PROGRAM ReactorLevelAndPressureController
VAR_INPUT
	serialCommData : ST_SerialCommReadData;
	stop : BOOL;
	levelHigh : BOOL;
END_VAR
VAR_OUTPUT
	slurryInletValve : BOOL;
	slurryOutletValve : BOOL;
	extractiveOutletOnOffValve : BOOL;
	extractiveOutletControlValveClose : BOOL;
	extractiveOutletControlValveOpen : BOOL;
END_VAR
VAR
	
	// Handlers to call
	HandlePressureSensorScaling : PressureSensorScalingHandler;
	HandleAutomaticExtraction : AutomaticExtractionHandler;
	HandleExtractiveOutlet : ExtractiveOutletHandler;

	_iPressureScaledValue: INT; //Scaled pressure value
	_bLevelControlSwitch : BOOL;
	_slurryInValveCommand : BOOL;
	_slurryOutValveCommand : BOOL;
	_pressureIntervals : ST_PressureIntervals;
	_extractiveControlValveCommands : ST_ExtractiveControlValveCommands;
	_ExtractiveControlValveParameters : ST_ExtractiveControlValveParameters;
	_automaticExtractionParameters : ST_AutomaticExtractionParameters;
	_decreasePumpSetpoint : BOOL;
	_controlValveOpening : DINT;
	_calibrateDone : BOOL;
	levelControlMode : INT;
	manualModeEntered : BOOL;
	autoModeEntered : BOOL;
	SlurryOutValveControl: FB_ReactorValves;
	sLevelControlState: STRING;
	sFillingValveState: STRING;;
	
	_extractiveOutOnOffValveCommand : BOOL;
	_startAutomaticExtraction : BOOL;
	
	_automaticExtractionState : E_AutomaticExtractionState;
	_automaticExtractionValues : ST_AutomaticExtractionValues;
	
	RTRIG_SetPressureReference : R_TRIG;
	pressureReference : INT;
	_extractiveOnOffValveValues : ST_ExtractiveOnOffValveValues;
END_VAR
VAR PERSISTENT
	_fillingValveOpenInterval: INT;
	_fillingValveCloseInterval: INT;	
END_VAR


HandlePressureSensorScaling(
						reactorPressureSensor := GVL_IO.reactorPressure,
						PressureScaledValue => _iPressureScaledValue);
						
HandleAutomaticExtraction(
						automaticExtractionParameters := _automaticExtractionParameters,
						extractiveControlValveParameters := _extractiveControlValveParameters,
						pressureScaledValue := _iPressureScaledValue,
						serialCommData := serialCommData,
						extractiveControlValveCommands := _extractiveControlValveCommands,
						pressureIntervals := _pressureIntervals,
						reactorLevelHigh := levelHigh,
						startAutomaticExtraction := _startAutomaticExtraction,
						calibrateDone := _calibrateDone,
						slurryInValveCommand := _slurryInValveCommand,
						slurryOutValveCommand := _slurryOutValveCommand ,
						decreasePumpSetpoint => _decreasePumpSetpoint,
						reactorInletValve => slurryInletValve,
						automaticExtractionState => _automaticExtractionState,
						extractiveOutOnOffValveAutoCommand => ,
						controlValveAutoOpenPercentage => ,
						reactorOutletValve => slurryOutletValve,
						automaticExtractionValues => _automaticExtractionValues);
						
HandleExtractiveOutlet(
					stop := stop,
					extractiveControlValveCommands := _ExtractiveControlValveCommands,
					extractiveControlValveParameters := _ExtractiveControlValveParameters,
					extractiveOutOnOffValveCommand := (_extractiveOutOnOffValveCommand AND (_automaticExtractionState = E_AutomaticExtractionState.MANUAL_EXTRACTION)) OR 
														((_automaticExtractionState <> E_AutomaticExtractionState.MANUAL_EXTRACTION) AND HandleAutomaticExtraction.extractiveOutOnOffValveAutoCommand),
					autoExtractionControlValveValue := HandleAutomaticExtraction.controlValveAutoOpenPercentage,
					autoExtractionStarted := _automaticExtractionState <> E_AutomaticExtractionState.MANUAL_EXTRACTION,
					controlValveOpeningPercentage => _controlValveOpening,
					extractiveOnOffValveValues => _extractiveOnOffValveValues,
					calibrateDone => _calibrateDone,
					openOnOffValve => extractiveOutletOnOffValve,
					closeExtractiveOutletValve => extractiveOutletControlValveClose,
					openExtractiveOutletValve => extractiveOutletControlValveOpen);

//IF _startAutomaticExtraction AND _calibrateDone THEN
//	manualModeEntered := FALSE;
	
//	// Automatic extraction
//	AutomaticExtraction(
//				parameters := _automaticExtractionParameters,
//				controlValveFullOpenTime := _ExtractiveControlValveParameters.timeToFullyOpenMs,
//				reactorPressure := _iPressureScaledValue,
//				pumpPressure := serialCommData.pumpingPressureMeasurement,
//				pumpSetpoint := SerialCommData.pumpingPressureSetpoint,
//				decreasePumpSetpoint => _decreasePumpSetpoint,
//				extractivePumpOn => GVL_IO.reactorInletValve,
//				co2onOffValveClosed => ,
//				automaticExtractionState => _automaticExtractionState);
//	_extractiveOutOnOffValveCommand := NOT AutomaticExtraction.co2onOffValveClosed;
//	_extractiveControlValveCommands.openPercentage := AutomaticExtraction.controlValveOpeningPercentage;
	
//	// Slurry outlet valve control
//	RTRIG_SetPressureReference(CLK := _automaticExtractionState = E_AutomaticExtractionState.FILLING_ACTIVE);
//	IF RTRIG_SetPressureReference.Q THEN
//		pressureReference :=  _iPressureScaledValue;
//	END_IF
//	SlurryOutValveControl.pressureIntervalControl(
//										interval_1_condition:= GVL_IO.reactorInletValve,// GVL_IO.reactorLevelHigh AND GVL_IO.reactorInletValve, // If above higher limit and filling valve open
//										pressureUpperInterval_1:= _pressureIntervals.PressureUpperInterval_1, 
//										pressureLowerInterval_1:= _pressureIntervals.PressureLowerInterval_1, 
//										interval_2_condition:= FALSE,//GVL_IO.reactorLevelHigh AND NOT GVL_IO.reactorInletValve,  // If above higher limit and filling valve closed
//										pressureUpperInterval_2:= _pressureIntervals.PressureUpperInterval_2, 
//										pressureLowerInterval_2:= _pressureIntervals.PressureLowerInterval_2, 
//										interval_3_condition:= FALSE,//NOT GVL_IO.reactorLevelHigh AND GVL_IO.reactorInletValve,  // If below higher limit and reactor filling valve open
//										pressureUpperInterval_3:= _pressureIntervals.PressureUpperInterval_3, 
//										pressureLowerInterval_3:= _pressureIntervals.PressureLowerInterval_3, 
//										pressureValue:= _iPressureScaledValue,  
//										pressureReference:= pressureReference,//_iPressureScaledValue,//DINT_TO_INT(SerialCommunicationHandler.pumpingPressureSetpoint), 
//										valveOpenCondition:= NOT (NOT GVL_IO.reactorLevelHigh AND NOT GVL_IO.reactorInletValve), 
//										forceValveClosed:= (NOT GVL_IO.reactorLevelHigh AND NOT GVL_IO.reactorInletValve),
//										);
//	GVL_IO.reactorOutletValve := SlurryOutValveControl.pressureControlOpen;
	
//ELSE
//	AutomaticExtraction.resetState();
//	// Close inlet/outlet valves when manual mode entered
//	IF NOT manualModeEntered THEN
//		GVL_IO.reactorInletValve := FALSE; // Close all valves when auto mode is exited
//		GVL_IO.reactorOutletValve := FALSE;
//		autoModeEntered := FALSE;
//		manualModeEntered := TRUE;
//	END_IF
//	GVL_IO.reactorInletValve := _slurryInValveCommand;
//	GVL_IO.reactorOutletValve := _slurryOutValveCommand;

//	_automaticExtractionState := E_AutomaticExtractionState.MANUAL_EXTRACTION;
	
//END_IF

//// Extractive outlet control
//_extractiveControlValveCommands.stopCalibration := Safety.stop;
//HandleExtractiveOutlet(
//					onOffValveCommand := _extractiveOutOnOffValveCommand,
//					controlValveCommands := _ExtractiveControlValveCommands,
//					controlValveParameters := _ExtractiveControlValveParameters,
//					onOffValveOpen => ,
//					onOffValveButtonCommand => GVL_IO.extractiveOutletOnOffValve,
//					controlValveClose => GVL_IO.extractiveOutletControlValveClose,
//					controlValveOpen => GVL_IO.extractiveOutletControlValveOpen,
//					controlValveCurrentOpenPercentage => _controlValveOpening,
//					calibrateDone => _calibrateDone);
//_extractiveOnOffValveValues.open := HandleExtractiveOutlet.onOffValveOpen;

PROPERTY AutomaticExtractionParameters : ST_AutomaticExtractionParameters
SET

_automaticExtractionParameters := AutomaticExtractionParameters;
END_SET
END_PROPERTY

PROPERTY automaticExtractionState : E_AutomaticExtractionState
GET

automaticExtractionState := _automaticExtractionSTate;
END_GET
END_PROPERTY

PROPERTY AutomaticExtractionValues : ST_AutomaticExtractionValues
GET

AutomaticExtractionValues := _automaticExtractionValues;
END_GET
END_PROPERTY

PROPERTY bLevelControlSwitch : BOOL
SET

_bLevelControlSwitch := bLevelControlSwitch;
END_SET
END_PROPERTY

PROPERTY CalibrateDone : BOOL
GET

CalibrateDone := _calibrateDone;
END_GET
END_PROPERTY

PROPERTY ControlValveOpening : DINT
GET

ControlValveOpening := _controlValveOpening;
END_GET
END_PROPERTY

PROPERTY controlValveOpeningOrClosing : BOOL
GET

controlValveOpeningOrClosing := GVL_IO.extractiveOutletControlValveClose OR GVL_IO.extractiveOutletControlValveOpen;
END_GET
END_PROPERTY

PROPERTY decreasePumpSetpoint : BOOL
GET

decreasePumpSetpoint := _decreasePumpSetpoint;
END_GET
END_PROPERTY

PROPERTY ExtractiveControlValveCommands : ST_ExtractiveControlValveCommands
SET
IF NOT _startAutomaticExtraction THEN
	_ExtractiveControlValveCommands := ExtractiveControlValveCommands;
END_IF
END_SET
END_PROPERTY

PROPERTY ExtractiveControlValveParameters : ST_ExtractiveControlValveParameters
SET

_ExtractiveControlValveParameters := ExtractiveControlValveParameters;
END_SET
END_PROPERTY

PROPERTY ExtractiveOnOffValveValues : ST_ExtractiveOnOffValveValues
GET

ExtractiveOnOffValveValues := _extractiveOnOffValveValues;
END_GET
END_PROPERTY

PROPERTY ExtractiveOutOnOffValveCommand : BOOL
SET

_extractiveOutOnOffValveCommand := ExtractiveOutOnOffValveCommand;
END_SET
END_PROPERTY

PROPERTY fillingValveCloseInterval : INT
SET

_fillingValveCloseInterval := fillingValveCloseInterval;
END_SET
END_PROPERTY

PROPERTY fillingValveOpenInterval : INT
SET

_fillingValveOpenInterval := fillingValveOpenInterval;
END_SET
END_PROPERTY

PROPERTY iPressureScaledValue : INT
GET

iPressureScaledValue := _iPressureScaledValue;
END_GET
END_PROPERTY

PROPERTY PressureIntervals : ST_PressureIntervals
SET

_pressureIntervals := PressureIntervals;
END_SET
END_PROPERTY

PROPERTY SlurryInValveCommand : BOOL
SET

_slurryInValveCommand := SlurryInValveCommand;
END_SET
END_PROPERTY

PROPERTY SlurryOutValveCommand : BOOL
SET

_slurryOutValveCommand := SlurryOutValveCommand;
END_SET
END_PROPERTY

PROPERTY StartAutomaticExtraction : BOOL
SET

_startAutomaticExtraction := StartAutomaticExtraction;
END_SET
END_PROPERTY

END_PROGRAM

(* stored: Version 1.1.0.1, ProductVersion 3.1.4024.9
   POU ReactorLevelAndPressureController: Id {a387b85d-f129-4119-abd4-456930450f01}, SpecialFunc None
   Property AutomaticExtractionParameters: Id {30db7c23-a067-400b-9e09-a227b67a6ab4}
   Set Set: Id {44547d4d-3b8d-4052-b809-8061fefc9dca}
   Property automaticExtractionState: Id {6405940a-3fdd-4150-8d77-d2c9ba3b9f2d}
   Get Get: Id {3dbfd90a-1f39-428e-a838-55a53fa67dba}
   Property AutomaticExtractionValues: Id {7f4d11a0-f795-4f71-802d-589f306f93a9}
   Get Get: Id {25ce779e-140f-4a83-8f99-8465573a1082}
   Property bLevelControlSwitch: Id {157d05c6-890c-4007-9267-879a33c29919}
   Set Set: Id {6f409d45-6c86-41c4-88fa-9adadc01cff5}
   Property CalibrateDone: Id {c583b2fd-ab10-4bad-a67c-458211bdff0b}
   Get Get: Id {b16d9464-4f0a-47ab-b2ca-64bc10567fdb}
   Property ControlValveOpening: Id {8b5489cb-a22f-43c6-aa77-e1d04d2a5ecc}
   Get Get: Id {5f05338c-9c74-4abb-8260-acdeabac824b}
   Property controlValveOpeningOrClosing: Id {2e4da57c-5e38-4d17-b858-c5f4b05dced5}
   Get Get: Id {dfc2ed8a-b3d1-4793-a5d8-2b1e0b6fabc0}
   Property decreasePumpSetpoint: Id {6a5e7efb-c62b-441b-a388-1d2e40f8fc87}
   Get Get: Id {f104881b-5ef5-4720-8f6f-a548a9c92c63}
   Property ExtractiveControlValveCommands: Id {1bfd9b44-c696-40f5-998c-868a11dbfb00}
   Set Set: Id {3bcffb92-b59c-43ce-bc66-fdc818ccc0ba}
   Property ExtractiveControlValveParameters: Id {bb956caa-eeb6-470f-a093-928f6c7d6265}
   Set Set: Id {4b282e61-efe3-4f89-8e8a-75e12ec61769}
   Property ExtractiveOnOffValveValues: Id {50523ea0-c94e-4846-a787-c1142eb03a88}
   Get Get: Id {c8c9e1ec-2584-42a6-9608-d5c9b20f91fd}
   Property ExtractiveOutOnOffValveCommand: Id {461a6a9f-281d-484c-948f-8a31cb53f17c}
   Set Set: Id {56f473f2-6b90-480e-9099-0f83e1c5bbdc}
   Property fillingValveCloseInterval: Id {6a88157e-ad1e-4b33-b420-23e077b392b3}
   Set Set: Id {ecae8a8d-2f82-4ab1-b797-5f8a6ba22e3e}
   Property fillingValveOpenInterval: Id {1a5a0701-ed7c-4ad0-b561-bf5a253bdcbd}
   Set Set: Id {c5a68f5f-e948-4258-ab24-2caf6453de2b}
   Property iPressureScaledValue: Id {f3fccc10-a324-4a46-aa67-2f5a5ade620e}
   Get Get: Id {b24340e3-e276-44cc-aedf-92fb116f5053}
   Property PressureIntervals: Id {590fbcd9-9ded-465e-b5f3-c87f976ee592}
   Set Set: Id {55337214-2fb9-445e-aa8b-e3a09f5ae5e0}
   Property SlurryInValveCommand: Id {cf2e99f8-1ae2-4412-8aaa-3a3f4953daac}
   Set Set: Id {fa7013a0-5634-4bfb-bf36-3d02e0323469}
   Property SlurryOutValveCommand: Id {28697755-784a-4676-838b-2343170d2384}
   Set Set: Id {b5d4a71f-8119-4ac2-95c8-c61337f36845}
   Property StartAutomaticExtraction: Id {4c252e86-25fd-4464-9210-a67f9c79854e}
   Set Set: Id {558b9670-5a88-4dbb-ad82-582bd57fdf34} *)
